(* IEC 61131-3 sources: plcc/tests/fixtures/typecheck, 3 files *)

(* ---- fb_instantiation.st ---- *)
FUNCTION_BLOCK Counter
VAR_INPUT
    reset : BOOL;
END_VAR
VAR_OUTPUT
    count : INT;
END_VAR
VAR
    cnt : INT := 0;
END_VAR
    IF reset THEN
        cnt := 0;
    ELSE
        cnt := cnt + 1;
    END_IF;
    count := cnt;
END_FUNCTION_BLOCK

PROGRAM UseCounter
VAR
    my_counter : Counter;
    result : INT;
END_VAR
    my_counter(reset := FALSE);
    result := my_counter.count;
END_PROGRAM

(* ---- implicit_conversions.st ---- *)
PROGRAM ImplicitConv
VAR
    s : SINT := 1;
    i : INT := 2;
    d : DINT := 3;
    r : REAL := 1.0;
    lr : LREAL := 2.0;
END_VAR
    i := s;
    d := i;
    r := i;
    lr := r;
END_PROGRAM

(* ---- type_errors.st ---- *)
PROGRAM TypeErrors
VAR
    b : BOOL;
    i : INT;
    r : REAL;
END_VAR
    i := b + i;
    r := 'hello';
END_PROGRAM
